TYPE ST_LoadingStation_InOuts :
STRUCT
	iBottleDetectionSensor AT %I*:INT;
END_STRUCT
END_TYPE

(* stored: Version 1.1.0.1, ProductVersion 3.1.4024.15
   DUT ST_LoadingStation_InOuts: Id {675a0f29-2949-4371-bd1a-150550b89c80} *)
